(* PLC project AHU-Project.project, CODESYS CODESYS V3.5 SP21 Patch 5 *)
(* stored: creationDateTime 2026-06-06T22:39:09.1863454, modificationDateTime 2026-06-06T19:12:37.3097521 *)

PROGRAM PLC_PRG_LD

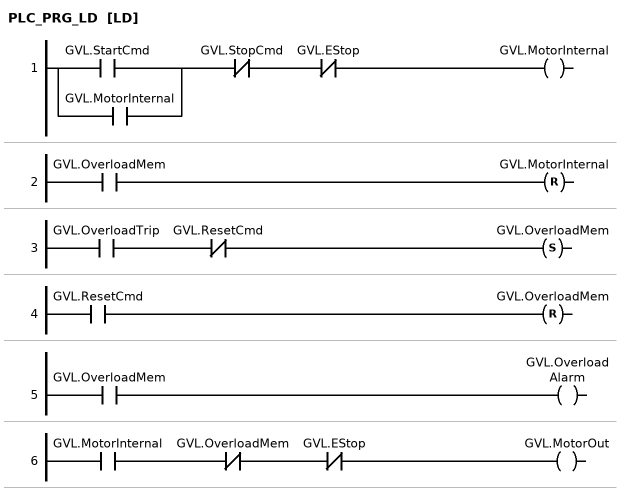
(* LD diagram, written out as Structured Text *)

GVL.MotorInternal := (GVL.StartCmd OR GVL.MotorInternal) AND NOT GVL.StopCmd AND NOT GVL.EStop;

IF GVL.OverloadMem THEN GVL.MotorInternal := FALSE; END_IF;

IF GVL.OverloadTrip AND NOT GVL.ResetCmd THEN GVL.OverloadMem := TRUE; END_IF;

IF GVL.ResetCmd THEN GVL.OverloadMem := FALSE; END_IF;

GVL.OverloadAlarm := GVL.OverloadMem;

GVL.MotorOut := GVL.MotorInternal AND NOT GVL.OverloadMem AND NOT GVL.EStop;
END_PROGRAM
